// TIA Portal project "FactoryIO_Template_S7-1200_V15_V15.1" (V15.1)
// Vorlageprojekt für das Buch mit Zielsystem S7-1200

(* hardware
DEVICE "S7-1200-Station_1"  S7-1200 Station
   slot 0: "Baugruppenträger_0"  Rack  V1.0
   slot 1: "PLC_1"  CPU 1211C DC/DC/DC  6ES7 211-1AE40-0XB0  V4.1
DEVICE "HMI_1"  KTP700 Basic PN
   slot 0: "HMI_1"  KTP700 Basic PN  6AV2 123-2GB03-0AX0  15.1.0.0
   slot 1: "HMI_RT_1"  KTP700 Basic PN  6AV2 123-2GB03-0AX0  15.1.0.0
   slot 5: "HMI_1.IE_CP_1"  PROFINET Interface  15.0.1.0
      slot 1: "PROFINET Interface_1"  PROFINET Interface
         slot 1: "Port_1"  Port
*)

// ===== PLC "PLC_1"  CPU 1211C DC/DC/DC =====

VAR_GLOBAL   // PLC tag table "Standard-Variablentabelle"
   "Tag_1" AT %A0.0 : Bool;
   "Tag_2" AT %E0.0 : Bool;
   "Tag_3" AT %E0.1 : Bool;
   "Tag_4" AT %QD30 : DWord;
END_VAR

VAR_GLOBAL   // PLC tag table "TAG_TABLE_FOR_IO"
   "Start" AT %I0.2 : Bool;   // Start Button
   "Stop" AT %I0.3 : Bool;   // Stop Button
   "Sensor1" AT %I0.4 : Bool;   // For Large box Sensor
   "Sensor2" AT %I0.5 : Bool;   // For small box Sensor
   "Pusher1" AT %Q0.1 : Bool;   // For Large box Pusher
   "Pusher2" AT %Q0.2 : Bool;   // For Large box Pusher
   "Conveyr1" AT %Q0.3 : Bool;
   "Conveyr2" AT %Q0.4 : Bool;
   "Conveyr3" AT %Q0.5 : Bool;
   "Conveyr4" AT %Q0.6 : Bool;
   "Red_Light" AT %Q0.7 : Bool;
   "Green_Light" AT %Q1.0 : Bool;
   "Conveyr5" AT %Q1.1 : Bool;
   "Reset1" AT %I1.0 : Bool;   // Counter Reset for Large Box
   "Reset2" AT %I1.1 : Bool;   // Counter Reset For Small Box
   "StackLightRed" AT %Q1.2 : Bool;
   "StackLightGreen" AT %Q1.3 : Bool;
   "First_Counter" AT %QW30 : Word;
   "Second_Counter" AT %QW34 : Word;
   "Conveyr6" AT %Q1.4 : Bool;
   "Emergency STOP" AT %I0.6 : Bool;
   "StartM" AT %M0.0 : Bool;
   "Conveyr7" AT %Q1.5 : Bool;
   "System Reset" AT %I1.2 : Bool;
   "FactorI0 Reset" AT %Q1.7 : Bool;
   "StackLightYellow" AT %Q1.6 : Bool;
END_VAR

// folder: System blocks/Program resources

DATA_BLOCK "IEC_Timer_0_DB"   // DB1
{ S7_Optimized_Access := 'TRUE' }
AUTHOR : Simatic
FAMILY : IEC
NAME : IEC_TMR
VERSION : 1.0
// stored: InstanceOfName IEC_TIMER
"IEC_TIMER"
BEGIN
END_DATA_BLOCK

DATA_BLOCK "IEC_Timer_0_DB_1"   // DB2
{ S7_Optimized_Access := 'TRUE' }
AUTHOR : Simatic
FAMILY : IEC
NAME : IEC_TMR
VERSION : 1.0
// stored: InstanceOfName IEC_TIMER
"IEC_TIMER"
BEGIN
END_DATA_BLOCK

DATA_BLOCK "IEC_Counter_0_DB_2"   // DB5
{ S7_Optimized_Access := 'TRUE' }
AUTHOR : Simatic
FAMILY : IEC
NAME : CNTR
VERSION : 1.0
// stored: InstanceOfName IEC_COUNTER
"IEC_COUNTER"
BEGIN
END_DATA_BLOCK

DATA_BLOCK "IEC_Counter_0_DB_3"   // DB6
{ S7_Optimized_Access := 'TRUE' }
AUTHOR : Simatic
FAMILY : IEC
NAME : CNTR
VERSION : 1.0
// stored: InstanceOfName IEC_COUNTER
"IEC_COUNTER"
BEGIN
END_DATA_BLOCK

// folder: (top level)

FUNCTION "MHJ-PLC-Lab-Function-S71200" : Void   // FC9000, SCL
{ S7_Optimized_Access := 'TRUE' }
VERSION : 0.1
   VAR_TEMP
      rdTimeReturn : Int;
      outputTime : DTL;
      SyncVal : Byte;
      forVal : Int;
      forVal_2 : Int;
      Value : Byte;
   END_VAR
   VAR CONSTANT
      CompVal : Byte := 16#34;
      Value_01 : Byte := 16#11;
      Value_01_DW : DWord := 16#A165_D992;
      Value_02_DW : DWord := 16#58BE_4401;
   END_VAR
BEGIN

   #Value:=PEEK(area := 16#82,
        dbNumber := 0,
        byteOffset := 511);
   #Value := #Value + 1;

   POKE(area := 16#82,
        dbNumber := 0,
        byteOffset := 511,
        value := #Value);

   POKE(area:=16#81,
        dbNumber:=0,
        byteOffset:=1016,
        value:=#Value_01_DW);
   POKE(area := 16#81,
        dbNumber := 0,
        byteOffset := 1020,
        value := #Value_02_DW);

   POKE(area := 16#81,
        dbNumber := 0,
        byteOffset := 511,
        value := B#16#00);

   FOR #forVal := 0 TO 120 DO
       FOR #forVal_2:=0 TO 10 DO
           #rdTimeReturn:=RD_SYS_T(#outputTime);
           #rdTimeReturn := WR_SYS_T(#outputTime);
           #rdTimeReturn := RD_SYS_T(#outputTime);
           #rdTimeReturn := WR_SYS_T(#outputTime);
       END_FOR;
       #SyncVal:= PEEK(area := 16#81,
                      dbNumber := 0,
                      byteOffset := 511);
       IF #SyncVal = #CompVal THEN
          GOTO M_1;
       END_IF;
   END_FOR;
   RETURN;

   M_1:
   POKE(area := 16#81,
        dbNumber := 0,
        byteOffset := 511,
        value := B#16#0);
END_FUNCTION

ORGANIZATION_BLOCK "Better_Not_To_Modify_This"   // OB1, FBD, ProgramCycle
TITLE = "Main Program Sweep (Cycle)"
{ S7_Optimized_Access := 'TRUE' }
VERSION : 0.1
   VAR_INPUT
      Initial_Call : Bool;   // Initial call of this OB
      Remanence : Bool;   // =True, if remanent data are available
   END_VAR
BEGIN

REGION Network 1: Konnektierungsbaustein für PLC-Lab
   // Im Netzwerk 1 wird der Konnektierungsbaustein für PLC-Lab aufgerufen.
   // Dieser Aufruf darf nicht entfernt werden!
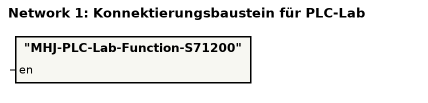
   "MHJ-PLC-Lab-Function-S71200"();
END_REGION

REGION Network 2: Ihr Programm
   // Schreiben Sie ab Netzwerk 2 Ihr Programm
END_REGION
END_ORGANIZATION_BLOCK

ORGANIZATION_BLOCK "Factory_IO_Control_Program"   // OB123, LAD, ProgramCycle
TITLE = "Main Program Sweep (Cycle)"
{ S7_Optimized_Access := 'TRUE' }
VERSION : 0.1
   VAR_INPUT
      Initial_Call : Bool;   // Initial call of this OB
      Remanence : Bool;   // =True, if remanent data are available
   END_VAR
BEGIN

REGION Network 1
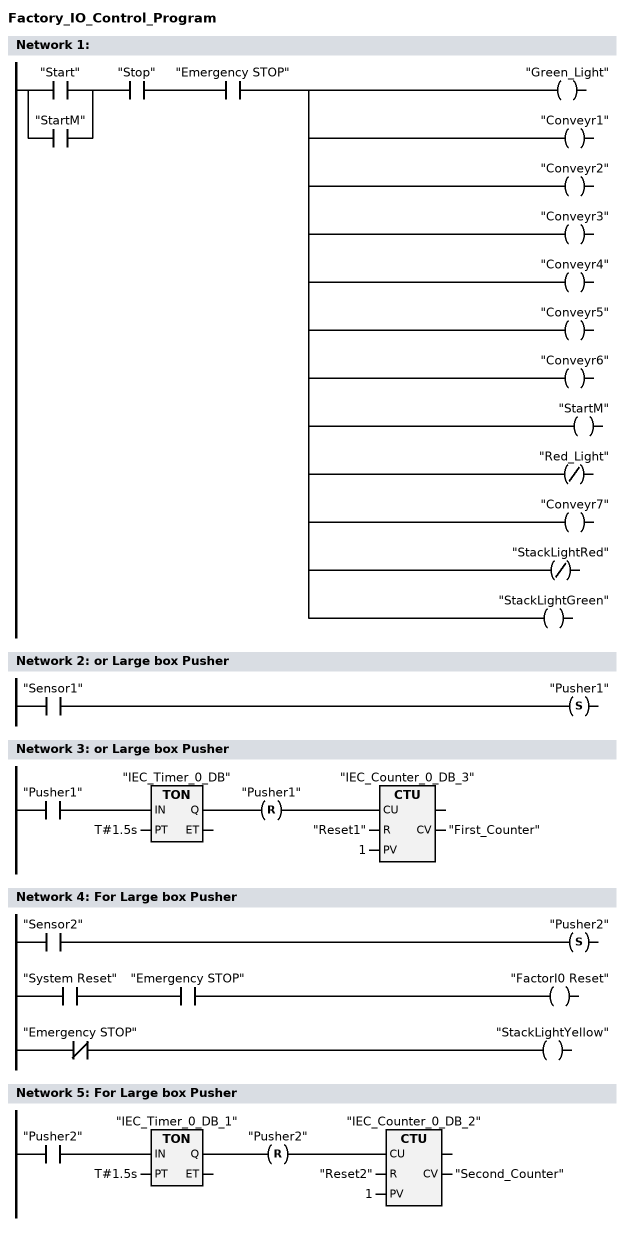
   RUNG wire#powerrail
      Contact( "Start" )
      wire#w1
      Contact( "Stop" )
      Contact( "Emergency STOP" )
      wire#w2
      Coil( "Green_Light" )
   END_RUNG
   RUNG wire#powerrail
      Contact( "StartM" )
   END_RUNG wire#w1
   RUNG wire#w2
      Coil( "Conveyr1" )
   END_RUNG
   RUNG wire#w2
      Coil( "Conveyr2" )
   END_RUNG
   RUNG wire#w2
      Coil( "Conveyr3" )
   END_RUNG
   RUNG wire#w2
      Coil( "Conveyr4" )
   END_RUNG
   RUNG wire#w2
      Coil( "Conveyr5" )
   END_RUNG
   RUNG wire#w2
      Coil( "Conveyr6" )
   END_RUNG
   RUNG wire#w2
      Coil( "StartM" )
   END_RUNG
   RUNG wire#w2
      I_Coil( "Red_Light" )
   END_RUNG
   RUNG wire#w2
      Coil( "Conveyr7" )
   END_RUNG
   RUNG wire#w2
      I_Coil( "StackLightRed" )
   END_RUNG
   RUNG wire#w2
      Coil( "StackLightGreen" )
   END_RUNG
   // the same network as SCL:
   "Green_Light" := ("Start" OR "StartM") AND "Stop" AND "Emergency STOP";
   "Conveyr1" := "Green_Light";
   "Conveyr2" := "Green_Light";
   "Conveyr3" := "Green_Light";
   "Conveyr4" := "Green_Light";
   "Conveyr5" := "Green_Light";
   "Conveyr6" := "Green_Light";
   "StartM" := "Green_Light";
   "Red_Light" := NOT "Green_Light";
   "Conveyr7" := "Green_Light";
   "StackLightRed" := NOT "Green_Light";
   "StackLightGreen" := "Green_Light";
END_REGION

REGION Network 2: or Large box Pusher
   RUNG wire#powerrail
      Contact( "Sensor1" )
      S_Coil( "Pusher1" )
   END_RUNG
   // the same network as SCL:
   IF "Sensor1" THEN "Pusher1" := TRUE; END_IF;
END_REGION

REGION Network 3: or Large box Pusher
   "IEC_Timer_0_DB".TON(IN := "Pusher1", PT := T#1.5s);
   IF "IEC_Timer_0_DB".Q THEN "Pusher1" := FALSE; END_IF;
   "IEC_Counter_0_DB_3".CTU(CU := "IEC_Timer_0_DB".Q, R := "Reset1", PV := 1, CV => "First_Counter");
END_REGION

REGION Network 4: For Large box Pusher
   RUNG wire#powerrail
      Contact( "Sensor2" )
      S_Coil( "Pusher2" )
   END_RUNG
   RUNG wire#powerrail
      Contact( "System Reset" )
      Contact( "Emergency STOP" )
      Coil( "FactorI0 Reset" )
   END_RUNG
   RUNG wire#powerrail
      I_Contact( "Emergency STOP" )
      Coil( "StackLightYellow" )
   END_RUNG
   // the same network as SCL:
   IF "Sensor2" THEN "Pusher2" := TRUE; END_IF;
   "FactorI0 Reset" := "System Reset" AND "Emergency STOP";
   "StackLightYellow" := NOT "Emergency STOP";
END_REGION

REGION Network 5: For Large box Pusher
   "IEC_Timer_0_DB_1".TON(IN := "Pusher2", PT := T#1.5s);
   IF "IEC_Timer_0_DB_1".Q THEN "Pusher2" := FALSE; END_IF;
   "IEC_Counter_0_DB_2".CTU(CU := "IEC_Timer_0_DB_1".Q, R := "Reset2", PV := 1, CV => "Second_Counter");
END_REGION
END_ORGANIZATION_BLOCK

(* ===== HMI "HMI_RT_1" =====
system functions are stored by id; their names below are inferred from use
connection "HMI_Connection_1": ETHERNET, SMART_S7_1200_OMS

HMI tags "Default tag table"
   "Tag_ScreenNumber" : UInt, internal
   "Start" : Bool = PLC Start AT %I0.2, 1 s
   "Stop" : Bool = PLC Stop AT %I0.3, 1 s
   "Reset1" : Bool = PLC Reset1 AT %I1.0, 1 s
   "Reset2" : Bool = PLC Reset2 AT %I1.1, 1 s
   "First_Counter" : Word = PLC First_Counter AT %QW30, 1 s
   "Second_Counter" : Word = PLC Second_Counter AT %QW34, 1 s
   "StartM" : Bool = PLC StartM AT %M0.0, 1 s
   "Emergency STOP" : Bool = PLC "Emergency STOP" AT %I0.6, 1 s
   "System Reset" : Bool = PLC "System Reset" AT %I1.2, 1 s

Template "Template_1" 800x480
   Button "Exit" at 714,429 size 71x50; TextOff 'Exit'; PictureOff "ExitRuntime_KTP700_Basic_PN_TR"; PictureOn "ExitRuntime_KTP700_Basic_PN_TR"
      on Release: StopRuntime(0)
   Button "Template_Button" at 614,429 size 71x50; TextOff 'Text'
   Button "Template_Button_1" at 514,429 size 71x50; TextOff 'Text'
   Button "Template_Button_2" at 414,429 size 71x50; TextOff 'Text'
   Button "Template_Button_3" at 314,429 size 71x50; TextOff 'Text'
   Button "Template_Button_4" at 214,429 size 71x50; TextOff 'Text'
   Button "Template_Button_5" at 114,429 size 71x50; TextOff 'Text'
   Button "Start screen" at 14,429 size 71x50; TextOff 'Start screen'; PictureOff "NavigateHome_KTP700_Basic_PN_TR"; PictureOn "NavigateHome_KTP700_Basic_PN_TR"
      on Release: ActivateScreen("Root screen", 0)
   SymbolicIOField "Symbolic_IO_Field_Screen" at 93,9 size 600x33; TextOff '0'; TextOn '1'; TextList "TextList_ScreenNames"
      ProcessValue <- "Tag_ScreenNumber"
      on Change: ActivateScreenByNumber("Tag_ScreenNumber", 0)
   DateTimeField "HmiScreenItemData" at 695,25 size 105x25
   DateTimeField "HmiScreenItemData_1" at 695,0 size 105x25
   GraphicView "Logo" at 0,0 size 91x51; Picture "Logo of HMI_1"

screen "Root screen" 800x480, template "Template_1"
   on GenerateScreen: SetTag("Start", 1)
   IOField "I/O field_1" at 527,192 size 153x68; FormatPattern 9999999999
      ProcessValue <- "Second_Counter"
   IOField "I/O field_2" at 349,192 size 152x68; FormatPattern 9999999999
      on Activate: SetBit(N)
      ProcessValue <- "First_Counter"
   Button "Button_1" at 150,196 size 96x32; TextOff 'START'
      on Press: function_b14e0dd5("Start", 0)
   Button "Button_2" at 150,238 size 96x32; TextOff 'STOP'
      on Press: function_b14e0dd5("Stop", 0)
   Button "Button_3" at 558,263 size 96x32; TextOff 'RESET'
      on Press: function_b14e0dd5("Reset2", 0)
   Button "Button_4" at 382,262 size 96x32; TextOff 'RESET'
      on Press: function_b14e0dd5("Reset1", 0)
   TextField "Text field_1" at 382,165 size 85x23; Text 'Big Boxes'
   TextField "Text field_2" at 550,169 size 104x23; Text 'Small Boxes'
   TextField "Text field_3" at 230,237 size 16x23; Text 'Text'
   Button "Button_5" at 8,56 size 194x32; TextOff 'EMERGENCY STOP'
      on Press: function_b14e0dd5("Emergency STOP", 0)
   Button "Button_6" at 355,84 size 344x52; TextOff 'Process'
      Appearance <- "StartM"
   Button "Button_7" at 10,102 size 192x33; TextOff 'System Reset'
      on Press: function_b14e0dd5("System Reset", 0)
*)